Staubli VAL3: Simulation.dtx

mdesc mNomSpeed
sio sSocket = {link=Socket\Feedback}
tool tToolSuccion = {z=110, fatherId=flange[0], ioLink=valve2}
num nConnection
num nRecvData
jointRx JApproach1 = {j2=9, j3=75, j5=93}
jointRx JHome = {j3=0.6}
screen sMonitor
num l_nRetVal
pointRx pApprBins = {x=488.533117374584, y=-4.31537939334066, z=79.7509349968276, rx=-179.999994995315, ry=-0.671274884561614, rz=0.0461961759228383, fatherId=world[0]}
pointRx pBinYellow = {x=537, y=-223, z=-169, ry=-180, rz=78, fatherId=world[0]}
pointRx pBinBlue = {x=537, y=-65, z=-169, ry=-180, rz=78, fatherId=world[0]}
pointRx pBinGreen = {x=537, y=80, z=-169, ry=-180, rz=78, fatherId=world[0]}
pointRx pBinBrown = {x=537, y=240, z=-169, ry=-180, rz=78, fatherId=world[0]}
jointRx jGetCinta = {j1=-85, j2=70, j3=55, j5=56}
bool bStop
num nkey
jointRx jAproachCinta = {j1=-82, j2=60, j3=56.5, j5=65}
pointRx pTable = {x=256.13, y=-12.37, z=-7.47, ry=-180, rz=0.046191606806918, fatherId=world[0]}
tool tToolGripper = {z=115, fatherId=flange[0], ioLink=valve1}
sio sPlc = {link=Socket\PLClient}
num nRecvPLC
